{attribute 'qualified_only'}
{attribute 'strict'}
TYPE EFeedbackMsgPsdChamber :
(
	InterlockPanelsMsg := 20,	
	SlitDoorPositionMsg := 30,
	SlitDoorOpenPositionMsg,
	SlitDoorClosePositionMsg,		
	CdaValveIsOpenMsg,
	RefreshingMsg
);
END_TYPE

(* stored: Version 1.1.0.1, ProductVersion 3.1.4024.12
   DUT EFeedbackMsgPsdChamber: Id {9b5ed334-ee3e-4914-95af-b96c5acfa33e} *)
